FUNCTION_BLOCK FB_Drive_control
VAR_INPUT
	Safety_interlock:BOOL;
	Torque_prediction:INT;
	Speed:INT; (*When this speed is exceeded, the winder will go from torque control to speed control*)
	Movement_detect:BOOL;
	Motor_fed:BOOL;
	Auto_run:BOOL;
	Auto_ref:INT;
	Auto_trail_brakes:BOOL;
	Speed_scale:INT; (*Full lever speed (modified by creep/slow switch*)
	Lh_allowed_speed:INT;
	Rh_allowed_speed:INT;
	Current_limit:INT; (*Current limit in Amps*)
	Max_lever_amps:INT; (*Current ramp rate in Amps*)
	Speed_ramp_rate:INT; (*Speed ramp rate (accel and decel) in mm/s.*)
	Current_ramp_rate:INT; (*Ramp rate of armature current reference in A/s used in torque control*)
	Armature_current:REAL; (*Armature current in Amps*)
	Forward_backout:BOOL;
	Reverse_backout:BOOL;
END_VAR
VAR_OUTPUT
	Enable:BOOL; (*Drive enable signal*)
	Start:BOOL; (*Drive start/run signal*)
	Speed_control:BOOL; (*Drive required to be in speed control*)
	Torque_control:BOOL; (*Drive required to be in torque control*)
	Field_weakening:BOOL; (*Field weakening request (for DC drive)*)
	Brake_release:BOOL;
	Trail_brakes:BOOL;
	Driver_ref_final:INT;
	Speed_ref:INT; (*Speed reference in mm/s*)
	Torque_ref:INT; (*Torque reference in amps*)
	Drive_speed_ref:REAL; (*Speed reference to drive scaled according to Speed_10V*)
	Drive_torque_ref:INT; (*Torque reference to drive scaled according to Torque_10V (bipolar)*)
	Combined_ref:INT; (*Speed and torque reference combined output (e.g. for TPD32/DCV104)*)
	No_start:BOOL;
	Stall:BOOL;
	Enable_vs_motor_fed:BOOL;
	hmi_data:dut_hmi_Drive_control;
END_VAR
VAR_IN_OUT
	Settings:dut_Drive_control;
	Mode:dut_Mode;
	Brakes:dut_Brake;
	Clutch:dut_Clutch;
	Power_lever:dut_Power_lever;
	Safety:dut_Safety;
END_VAR
VAR
	R_TRIG_0: R_TRIG;
	RS_0: RS;
	Torq_ctl_brakes_on: BOOL;
	TON_0: TON;
	Kill_torq_ctl: BOOL;
	RS_1: RS;
	RS_2: RS;
	Lincon_0: FB_Lincon;
	Allowed_speed: INT;
	Ref_ramp_0: FB_Ref_ramp;
	Ref_ramp_1: FB_Ref_ramp;
	Torque_prediction_ramp: REAL;
	Lincon_1: FB_Lincon;
	Ref_ramp_2: FB_Ref_ramp;
	Lincon_2: FB_Lincon;
	Lincon_3: FB_Lincon;
	Manual_enable: BOOL;
	Auto_enable: BOOL;
	TON_1: TON;
	Safe_to_lift_brakes: BOOL;
	Lincon_4: FB_Lincon;
	Lincon_5: FB_Lincon;
	Pos_torque: BOOL;
	TON_2: TON;
	RS_3: RS;
	TON_3: TON;
	TON_4: TON;
	TON_5: TON;
	BIT_TO_WORD_V0_0: FB_BIT_TO_WORD_V0;
END_VAR

M_Torque_control();
M_Speed_scale();
M_Speed_ref();
M_Torque_ref();
M_Drive_references();
M_Drive_control();
M_Brake_control();
M_Trips();
M_HMI_data();

METHOD M_Brake_control
VAR_INPUT
END_VAR

VAR
END_VAR
VAR_INST // added by the converter: edge detectors and wires of the graphical bodies
    _w1, _w2, _w5, _w6, _w7, _w8, _w9, _w11, _w12, _w13 : BOOL;
    _w3, _w4, _w10 : ANY;
END_VAR
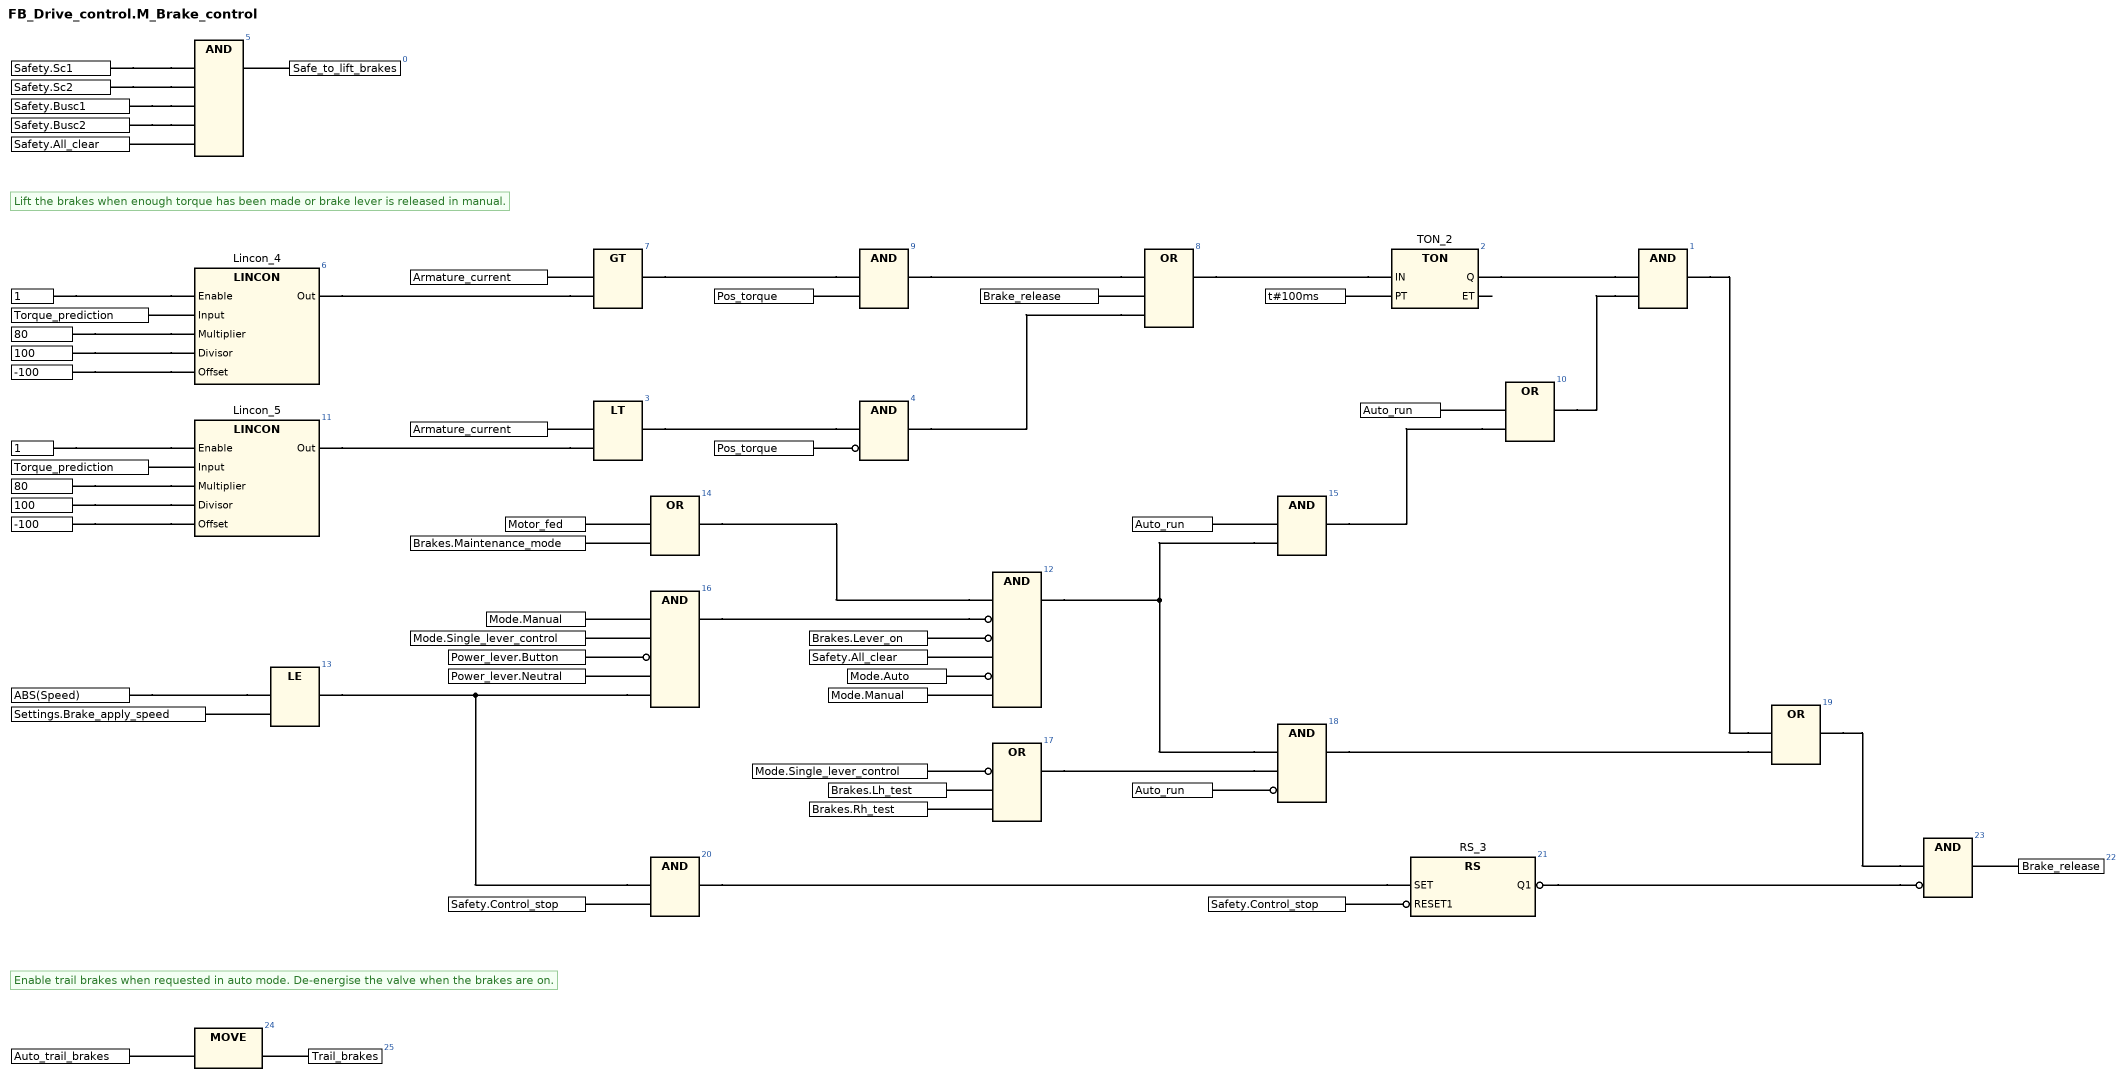
Safe_to_lift_brakes := _w1;
_w3 := TON_2.Q AND _w2;
TON_2(IN := _w4, PT := t#100ms); // TON
_w5 := Armature_current < Lincon_5.Out AND NOT Pos_torque;
_w1 := Safety.Sc1 AND Safety.Sc2 AND Safety.Busc1 AND Safety.Busc2 AND Safety.All_clear;
// Lift the brakes when enough torque has been made or brake lever is released in manual.
Lincon_4(Enable := 1, Input := Torque_prediction, Multiplier := 80, Divisor := 100, Offset := -100); // LINCON
_w4 := _w6 OR Brake_release OR _w5;
_w6 := Armature_current > Lincon_4.Out AND Pos_torque;
_w2 := Auto_run OR _w7;
Lincon_5(Enable := 1, Input := Torque_prediction, Multiplier := 80, Divisor := 100, Offset := -100); // LINCON
_w10 := _w8 AND NOT _w9 AND NOT Brakes.Lever_on AND Safety.All_clear AND NOT Mode.Auto AND Mode.Manual;
_w11 := (ABS(Speed)) <= Settings.Brake_apply_speed;
_w8 := Motor_fed OR Brakes.Maintenance_mode;
_w7 := Auto_run AND _w10;
_w9 := Mode.Manual AND Mode.Single_lever_control AND NOT Power_lever.Button AND Power_lever.Neutral AND _w11;
_w12 := _w3 OR _w10 AND (NOT Mode.Single_lever_control OR Brakes.Lh_test OR Brakes.Rh_test) AND NOT Auto_run;
RS_3(SET := _w11 AND Safety.Control_stop, RESET1 := NOT Safety.Control_stop); // RS
Brake_release := _w13;
_w13 := _w12 AND NOT (NOT RS_3.Q1);
// Enable trail brakes when requested in auto mode. De-energise the valve when the brakes are on.
Trail_brakes := Auto_trail_brakes;
END_METHOD

METHOD M_Drive_control
VAR_INPUT
END_VAR

VAR
END_VAR
VAR_INST // added by the converter: edge detectors and wires of the graphical bodies
    _w1, _w2, _w3, _w4, _w5, _w7, _w8, _w9, _w10, _w11 : BOOL;
    _w6 : ANY;
END_VAR
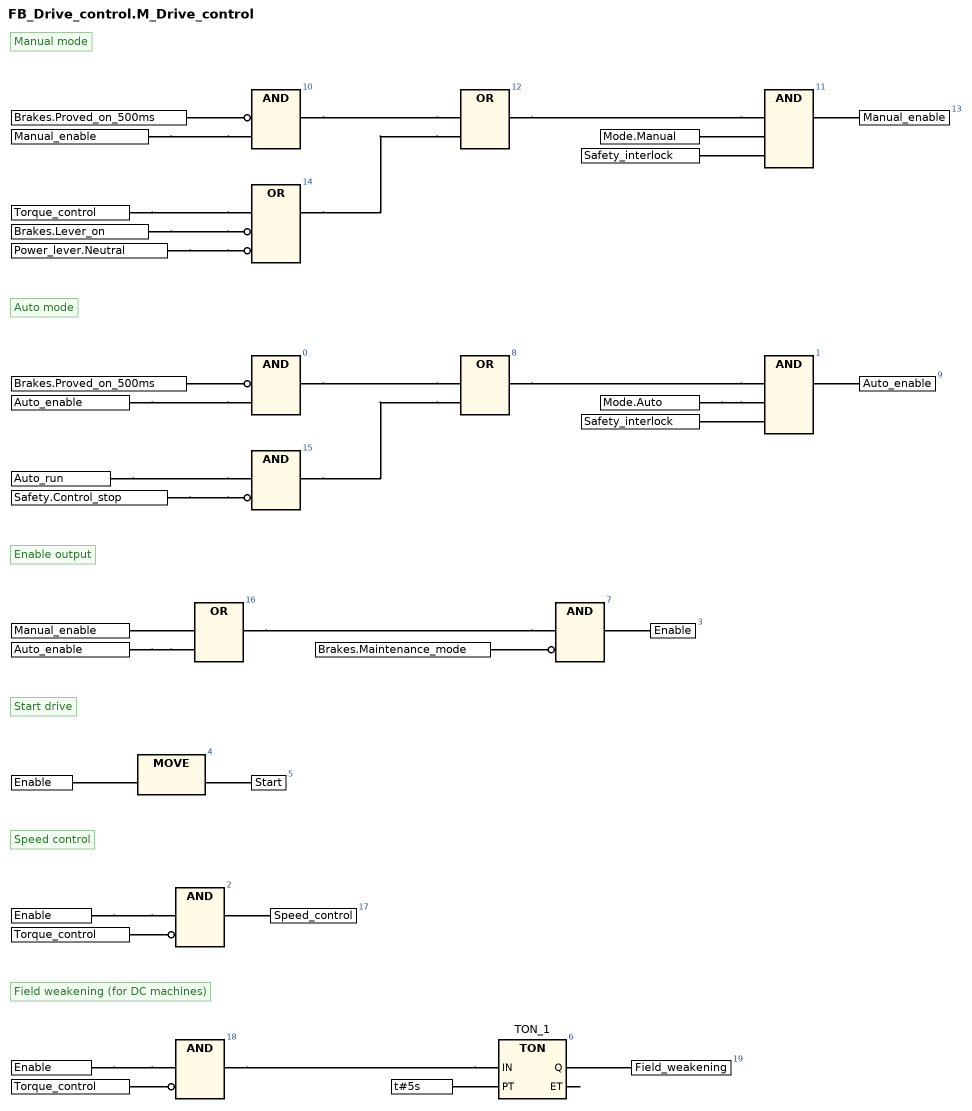
// Auto mode
_w1 := NOT Brakes.Proved_on_500ms AND Auto_enable;
_w3 := _w2 AND Mode.Auto AND Safety_interlock;
// Speed control
_w4 := Enable AND NOT Torque_control;
Enable := _w5;
// Start drive
Start := Enable;
TON_1(IN := _w6, PT := t#5s); // TON
_w5 := _w7 AND NOT Brakes.Maintenance_mode;
_w2 := _w1 OR _w8;
Auto_enable := _w3;
// Manual mode
_w10 := _w9 AND Mode.Manual AND Safety_interlock;
_w9 := NOT Brakes.Proved_on_500ms AND Manual_enable OR _w11;
Manual_enable := _w10;
_w11 := Torque_control OR NOT Brakes.Lever_on OR NOT Power_lever.Neutral;
_w8 := Auto_run AND NOT Safety.Control_stop;
// Enable output
_w7 := Manual_enable OR Auto_enable;
Speed_control := _w4;
// Field weakening (for DC machines)
_w6 := Enable AND NOT Torque_control;
Field_weakening := TON_1.Q;
END_METHOD

METHOD M_Drive_references
VAR_INPUT
END_VAR

VAR
	Drive_abs_torque: REAL;
	Pos_torque: BOOL;
END_VAR
VAR_INST // added by the converter: edge detectors and wires of the graphical bodies
    _w1 : INT;
    _w2 : REAL;
END_VAR
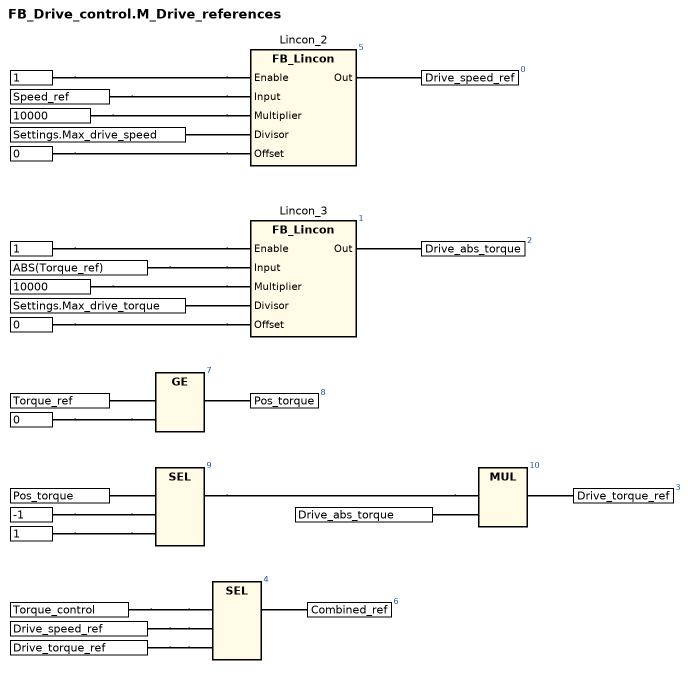
Drive_speed_ref := Lincon_2.Out;
Lincon_3(
    Enable := 1,
    Input := ABS(Torque_ref),
    Multiplier := 10000,
    Divisor := Settings.Max_drive_torque,
    Offset := 0); // FB_Lincon
Drive_abs_torque := Lincon_3.Out;
Drive_torque_ref := _w1;
_w2 := SEL(Torque_control, Drive_speed_ref, Drive_torque_ref);
Lincon_2(
    Enable := 1,
    Input := Speed_ref,
    Multiplier := 10000,
    Divisor := Settings.Max_drive_speed,
    Offset := 0); // FB_Lincon
Combined_ref := _w2;
Pos_torque := Torque_ref >= 0;
_w1 := SEL(Pos_torque, -1, 1) * Drive_abs_torque;
END_METHOD

METHOD M_HMI_data
VAR_INPUT
END_VAR
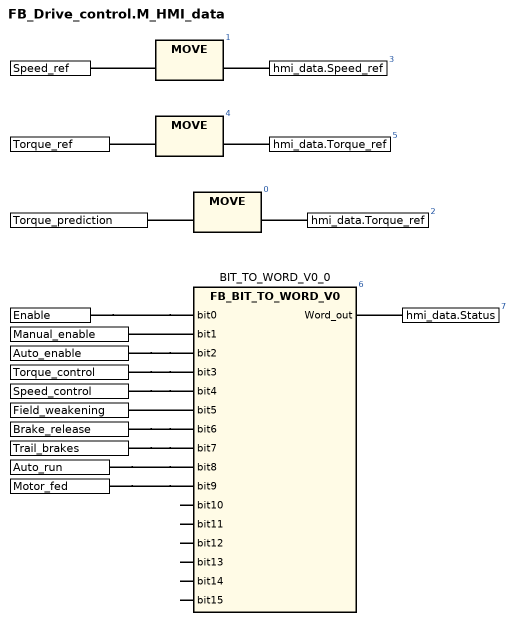
hmi_data.Torque_ref := Torque_prediction;
hmi_data.Speed_ref := Speed_ref;
hmi_data.Torque_ref := Torque_ref;
BIT_TO_WORD_V0_0(
    bit0 := Enable,
    bit1 := Manual_enable,
    bit2 := Auto_enable,
    bit3 := Torque_control,
    bit4 := Speed_control,
    bit5 := Field_weakening,
    bit6 := Brake_release,
    bit7 := Trail_brakes,
    bit8 := Auto_run,
    bit9 := Motor_fed); // FB_BIT_TO_WORD_V0
hmi_data.Status := BIT_TO_WORD_V0_0.Word_out;
END_METHOD

METHOD M_Speed_ref
VAR_INPUT
END_VAR

VAR
	
END_VAR
VAR_INST // added by the converter: edge detectors and wires of the graphical bodies
    _w1, _w3, _w4, _w5, _w6, _w7 : ANY;
    _w2 : INT;
END_VAR
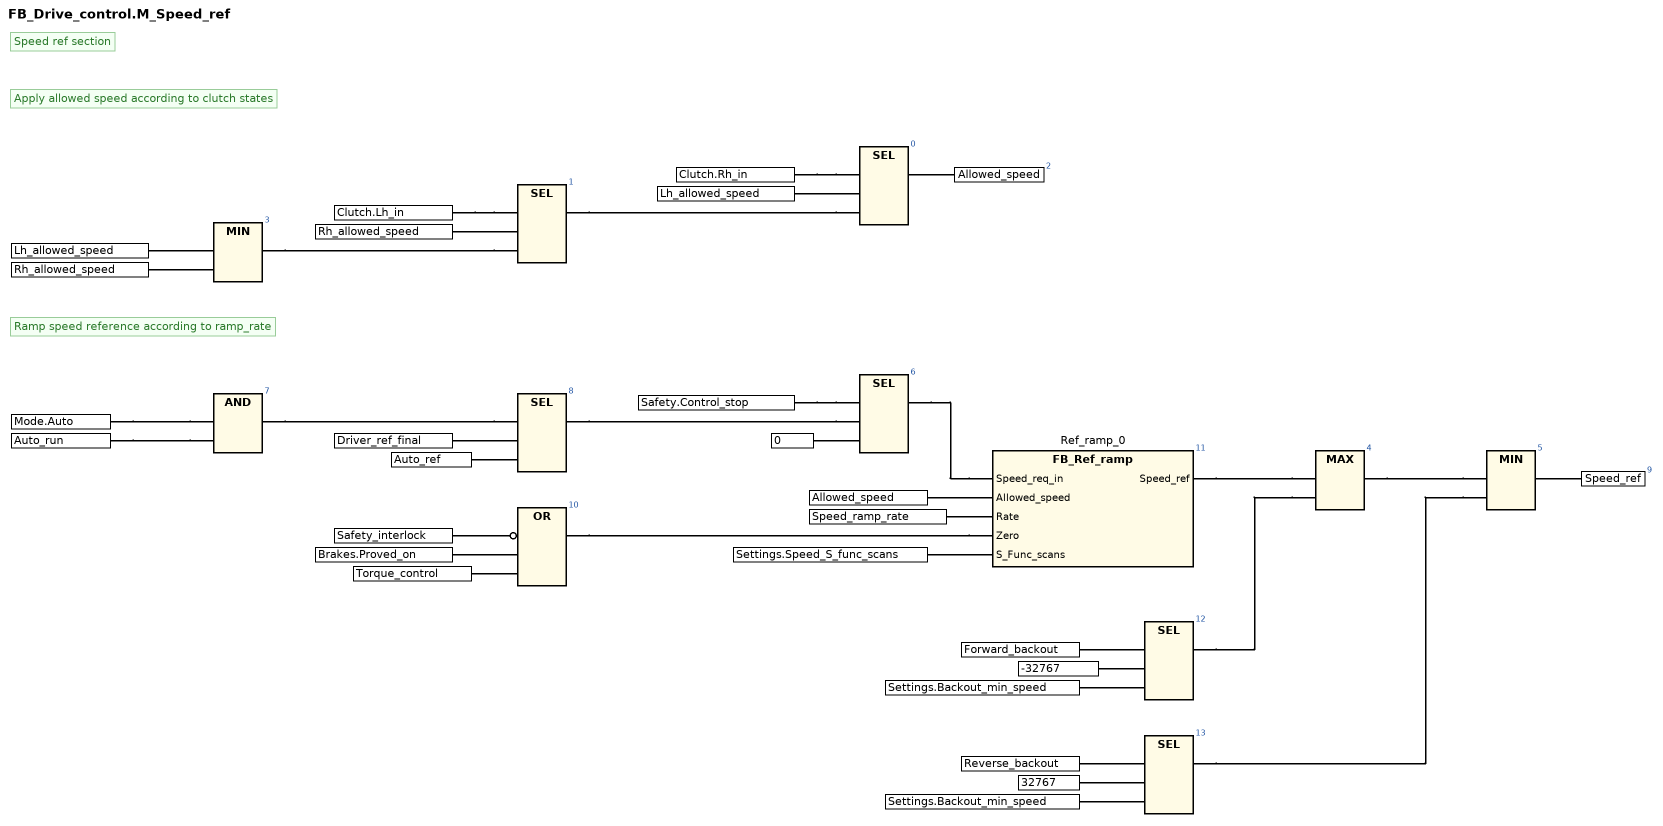
_w2 := SEL(Clutch.Rh_in, Lh_allowed_speed, _w1);
_w1 := SEL(Clutch.Lh_in, Rh_allowed_speed, _w3);
Allowed_speed := _w2;
// Speed ref section
// Apply allowed speed according to clutch states
_w3 := MIN(Lh_allowed_speed, Rh_allowed_speed);
_w7 := SEL(Safety.Control_stop, _w6, 0);
// Ramp speed reference according to ramp_rate
_w6 := SEL(Mode.Auto AND Auto_run, Driver_ref_final, Auto_ref);
Speed_ref := MIN(MAX(Ref_ramp_0.Speed_ref, _w4), _w5);
Ref_ramp_0(
    Speed_req_in := _w7,
    Allowed_speed := Allowed_speed,
    Rate := Speed_ramp_rate,
    Zero := NOT Safety_interlock OR Brakes.Proved_on OR Torque_control,
    S_Func_scans := Settings.Speed_S_func_scans); // FB_Ref_ramp
_w4 := SEL(Forward_backout, -32767, Settings.Backout_min_speed);
_w5 := SEL(Reverse_backout, 32767, Settings.Backout_min_speed);
END_METHOD

METHOD M_Speed_scale
VAR_INPUT
END_VAR
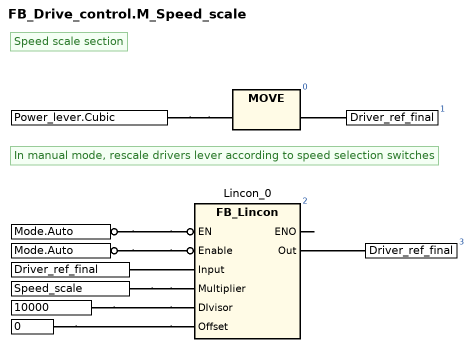
// Speed scale section
Driver_ref_final := Power_lever.Cubic;
// In manual mode, rescale drivers lever according to speed selection switches
IF NOT (NOT Mode.Auto) THEN
    Lincon_0(
        Enable := NOT (NOT Mode.Auto),
        Input := Driver_ref_final,
        Multiplier := Speed_scale,
        DIvisor := 10000,
        Offset := 0); // FB_Lincon
END_IF
Driver_ref_final := Lincon_0.Out;
END_METHOD

METHOD M_Torque_control
VAR_INPUT
END_VAR
VAR_INST // added by the converter: edge detectors and wires of the graphical bodies
    _w1, _w2, _w3, _w4, _w5, _w6, _w7 : BOOL;
END_VAR
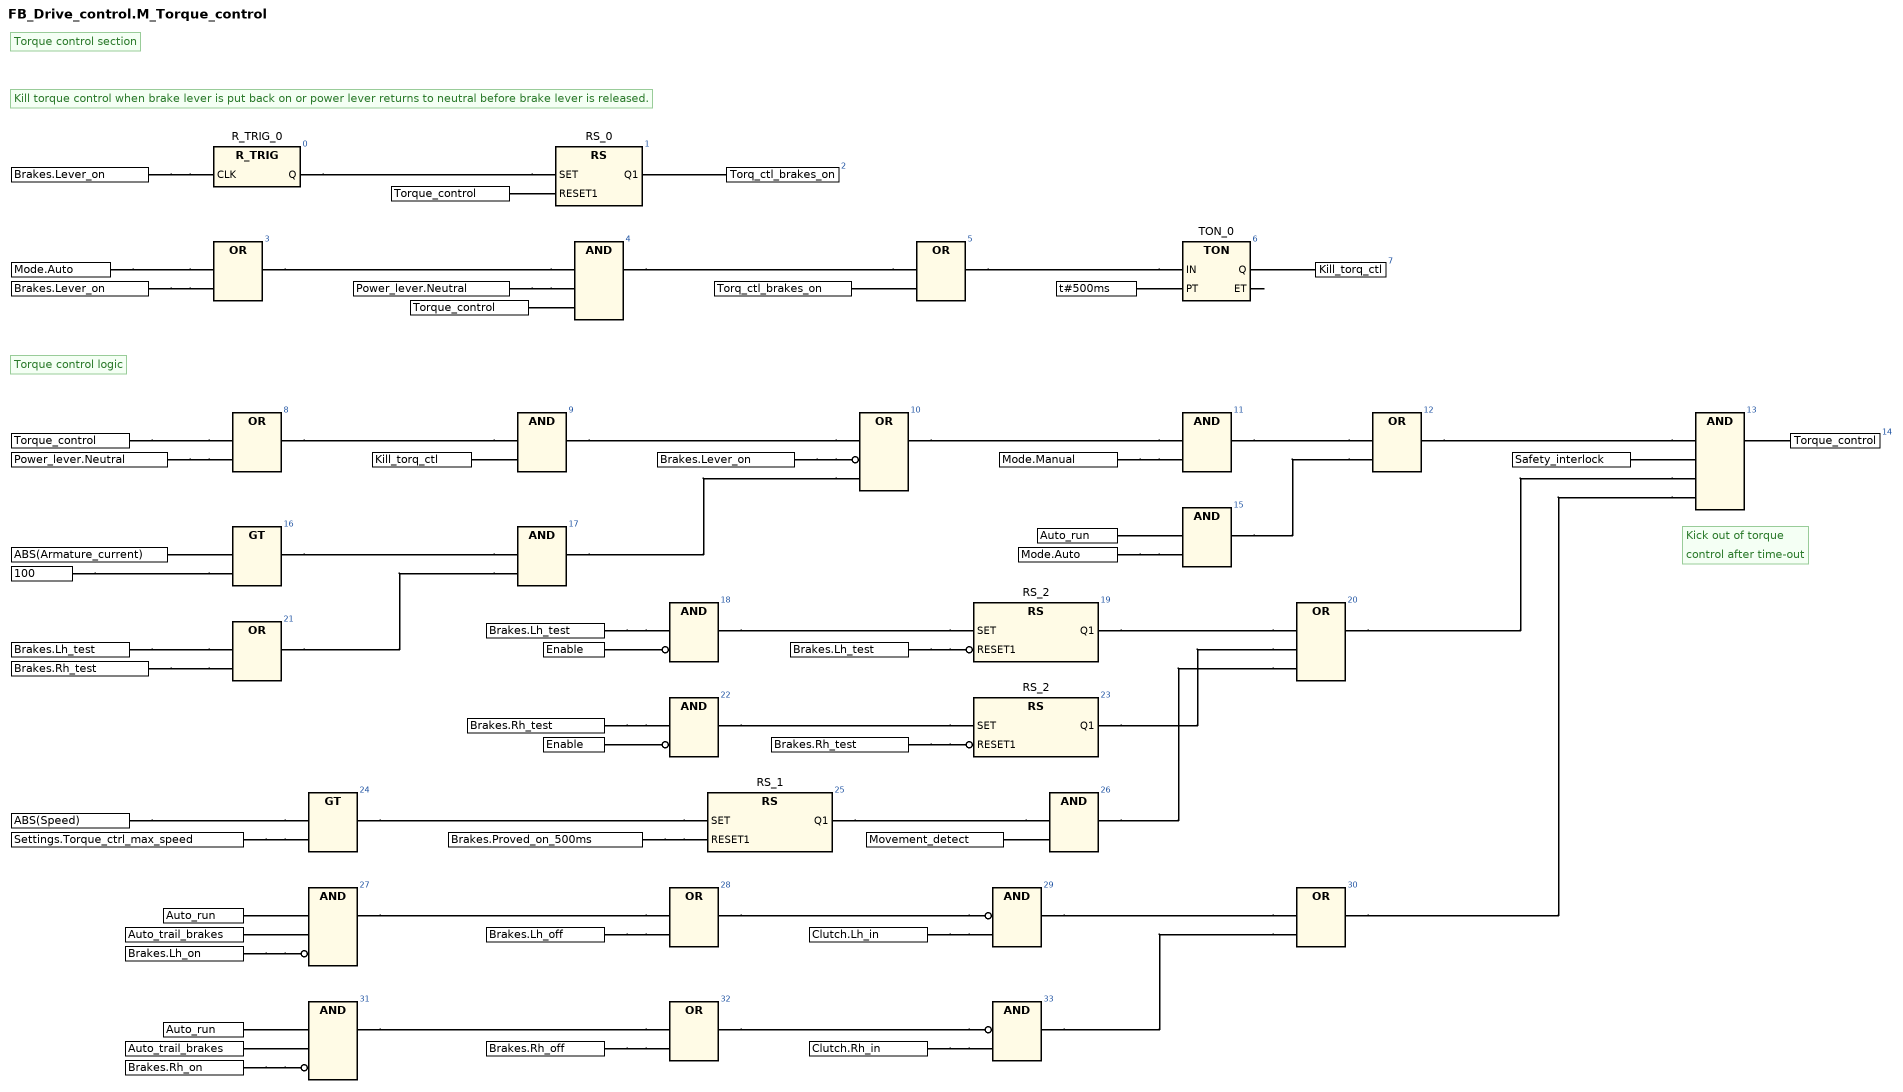
// Torque control section
// Kill torque control when brake lever is put back on or power lever returns to neutral before brake lever is released.
R_TRIG_0(CLK := Brakes.Lever_on); // R_TRIG
RS_0(SET := R_TRIG_0.Q, RESET1 := Torque_control); // RS
Torq_ctl_brakes_on := RS_0.Q1;
TON_0(IN := (Mode.Auto OR Brakes.Lever_on) AND Power_lever.Neutral AND Torque_control OR Torq_ctl_brakes_on, PT := t#500ms); // TON
Kill_torq_ctl := TON_0.Q;
// Torque control logic
Torque_control := (((Torque_control OR Power_lever.Neutral) AND Kill_torq_ctl OR NOT Brakes.Lever_on OR _w1) AND Mode.Manual OR _w2) AND Safety_interlock AND _w3 AND _w4;
_w2 := Auto_run AND Mode.Auto;
_w1 := (ABS(Armature_current)) > 100 AND _w5;
RS_2(SET := Brakes.Lh_test AND NOT Enable, RESET1 := NOT Brakes.Lh_test); // RS
// Kick out of torque
// control after time-out
_w3 := RS_2.Q1 OR RS_2.Q1 OR _w6;
_w5 := Brakes.Lh_test OR Brakes.Rh_test;
RS_2(SET := Brakes.Rh_test AND NOT Enable, RESET1 := NOT Brakes.Rh_test); // RS
RS_1(SET := (ABS(Speed)) > Settings.Torque_ctrl_max_speed, RESET1 := Brakes.Proved_on_500ms); // RS
_w6 := RS_1.Q1 AND Movement_detect;
_w4 := NOT (Auto_run AND Auto_trail_brakes AND NOT Brakes.Lh_on OR Brakes.Lh_off) AND Clutch.Lh_in OR _w7;
_w7 := NOT (Auto_run AND Auto_trail_brakes AND NOT Brakes.Rh_on OR Brakes.Rh_off) AND Clutch.Rh_in;
END_METHOD

METHOD M_Torque_ref
VAR_INPUT
END_VAR

VAR
END_VAR
VAR_INST // added by the converter: edge detectors and wires of the graphical bodies
    _w1 : INT;
    _w2, _w3, _w4, _w6, _w7, _w9, _w10 : ANY;
    _w5, _w8 : BOOL;
END_VAR
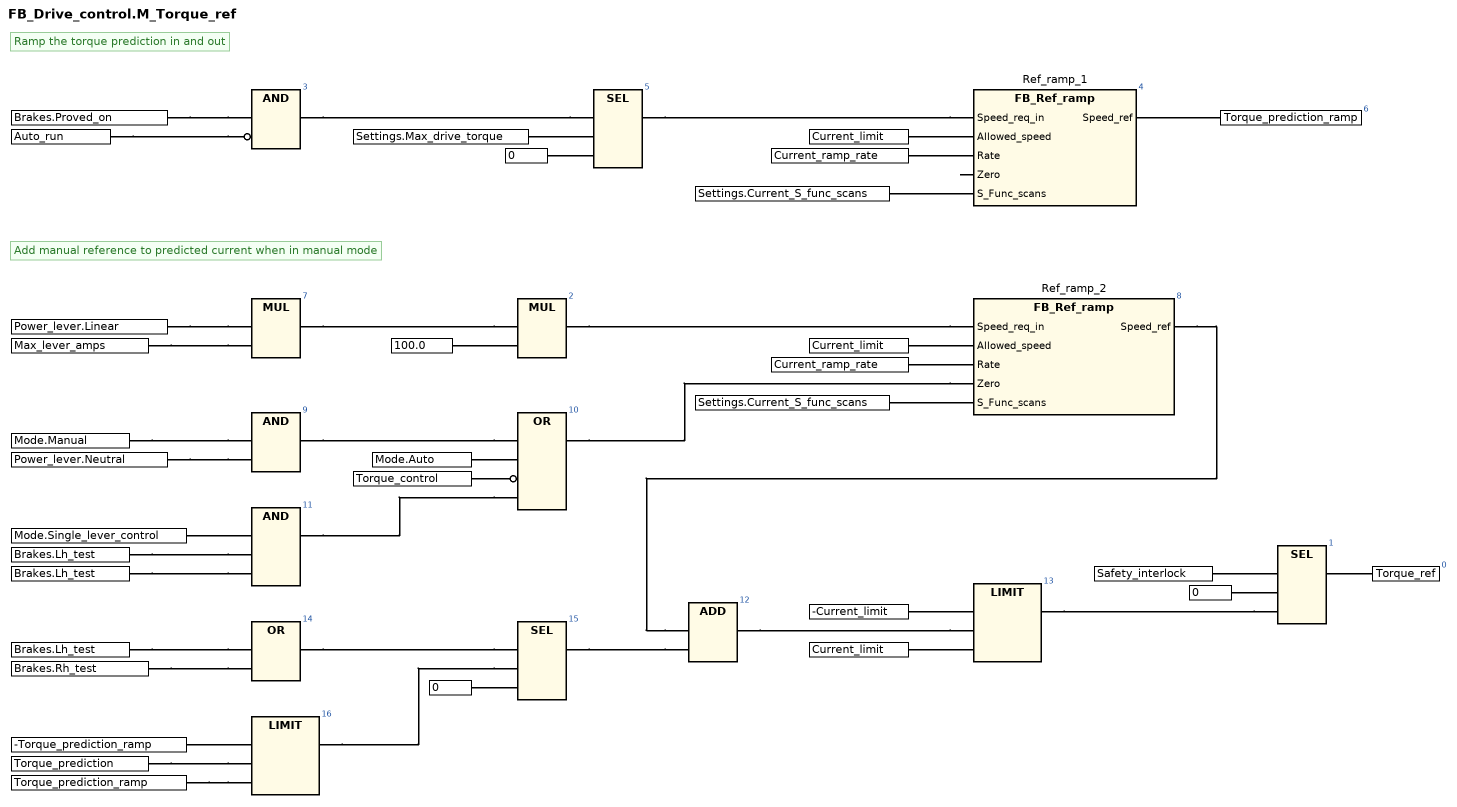
Torque_ref := _w1;
_w1 := SEL(Safety_interlock, 0, _w2);
_w4 := _w3 * 100.0;
// Ramp the torque prediction in and out
_w5 := Brakes.Proved_on AND NOT Auto_run;
Ref_ramp_1(
    Speed_req_in := _w6,
    Allowed_speed := Current_limit,
    Rate := Current_ramp_rate,
    S_Func_scans := Settings.Current_S_func_scans); // FB_Ref_ramp
_w6 := SEL(_w5, Settings.Max_drive_torque, 0);
Torque_prediction_ramp := Ref_ramp_1.Speed_ref;
// Add manual reference to predicted current when in manual mode
_w3 := Power_lever.Linear * Max_lever_amps;
Ref_ramp_2(
    Speed_req_in := _w4,
    Allowed_speed := Current_limit,
    Rate := Current_ramp_rate,
    Zero := _w7,
    S_Func_scans := Settings.Current_S_func_scans); // FB_Ref_ramp
_w7 := Mode.Manual AND Power_lever.Neutral OR Mode.Auto OR NOT Torque_control OR _w8;
_w8 := Mode.Single_lever_control AND Brakes.Lh_test AND Brakes.Lh_test;
_w2 := LIMIT(-Current_limit, Ref_ramp_2.Speed_ref + _w9, Current_limit);
_w9 := SEL(Brakes.Lh_test OR Brakes.Rh_test, _w10, 0);
_w10 := LIMIT(-Torque_prediction_ramp, Torque_prediction, Torque_prediction_ramp);
END_METHOD

METHOD M_Trips
VAR_INPUT
END_VAR
VAR_INST // added by the converter: edge detectors and wires of the graphical bodies
    _w1, _w3, _w5 : BOOL;
    _w2, _w4 : ANY;
END_VAR
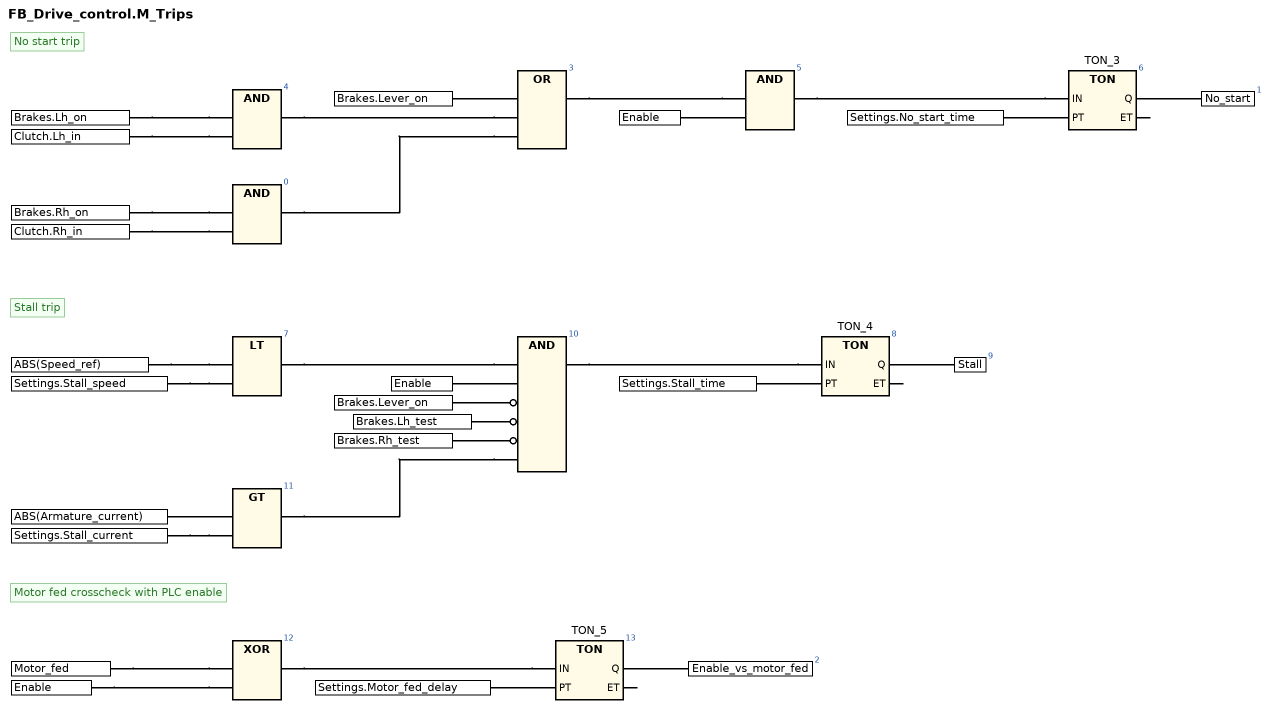
No_start := TON_3.Q;
Enable_vs_motor_fed := TON_5.Q;
_w2 := Brakes.Lever_on OR _w1 OR Brakes.Rh_on AND Clutch.Rh_in;
// No start trip
_w1 := Brakes.Lh_on AND Clutch.Lh_in;
TON_3(IN := _w2 AND Enable, PT := Settings.No_start_time); // TON
// Stall trip
_w3 := (ABS(Speed_ref)) < Settings.Stall_speed;
TON_4(IN := _w4, PT := Settings.Stall_time); // TON
Stall := TON_4.Q;
_w4 := _w3 AND Enable AND NOT Brakes.Lever_on AND NOT Brakes.Lh_test AND NOT Brakes.Rh_test AND _w5;
_w5 := (ABS(Armature_current)) > Settings.Stall_current;
// Motor fed crosscheck with PLC enable
TON_5(IN := Motor_fed XOR Enable, PT := Settings.Motor_fed_delay); // TON
END_METHOD

END_FUNCTION_BLOCK

(* stored: Version 1.1.0.1, ProductVersion 3.1.4024.0
   POU FB_Drive_control: Id {b4a159ff-53f5-4aca-a809-ec7186bb5eaa}, SpecialFunc None
   Method M_Brake_control: Id {5b486a7e-2a3d-4c9a-8ced-dc43c2f67684}
   Method M_Drive_control: Id {e907ed43-2ca4-489d-be3d-3cc06a104977}
   Method M_Drive_references: Id {79b8d2da-8e68-4ce1-874d-4ffcae92983e}
   Method M_HMI_data: Id {65165bf5-e0ec-40b6-b5f4-2f59f92d0484}
   Method M_Speed_ref: Id {49eb6c64-42aa-4def-9e6f-bf10a27ffbae}
   Method M_Speed_scale: Id {43cb51a1-2c09-4d26-9e1d-cfe32f140a17}
   Method M_Torque_control: Id {8864dd10-9af0-4e68-8028-7cd2a74a6d35}
   Method M_Torque_ref: Id {75215c45-8ea4-4495-a670-e9eac06b6975}
   Method M_Trips: Id {24338fdd-7a32-46f4-8bc3-ac8c36e24d51} *)
